ABB RobotStudio station: SemesterProjekt_sim_20200222-211423.rsstn

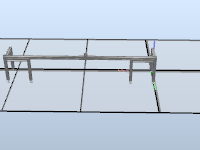
Station SemesterProjekt_sim (saved by RobotStudio 7.0.8728.594)
Layout (positions relative to the parent item):
  - BaseConstruktion [part] at (-0.03, 0.43, 41.45) mm, rotated rx 89.99 ry 0 rz -0.01 deg
  - Cart [part] at (558.99, 109.43, 431.44) mm, rotated rx 89.99 ry 0 rz -0.01 deg
  - endBlock [part] at (0, -450, 0) mm, rotated rx 90 ry 0 rz 0 deg
  - Part_7 [part] at (2080, 325.44, 436.4) mm, rotated rx 0 ry 0 rz 90 deg
  - Part_8 [part] at (40, 325.44, 436.4) mm, rotated rx 0 ry 0 rz 90 deg
